(* IEC 61131-3 sources: AXOpen/src/components.dukane.welders/ctrl/src/Axo_IQ_SeriesWelder (part 4) *)

            array_buffer[169].%X0 := buf5.LimitWeld1EnergyEnable._8;
            array_buffer[169].%X1 := buf5.LimitWeld1EnergyEnable._9;
            array_buffer[169].%X2 := buf5.LimitWeld1EnergyEnable._10;
            array_buffer[169].%X3 := buf5.LimitWeld1EnergyEnable._11;
            array_buffer[169].%X4 := buf5.LimitWeld1EnergyEnable._12;
            array_buffer[169].%X5 := buf5.LimitWeld1EnergyEnable._13;
            array_buffer[169].%X6 := buf5.LimitWeld1EnergyEnable._14;
            array_buffer[169].%X7 := buf5.LimitWeld1EnergyEnable._15;

            array_buffer[170].%X0 := buf5.LimitWeld1EnergyEnable._16;
            array_buffer[170].%X1 := buf5.LimitWeld1EnergyEnable._17;
            array_buffer[170].%X2 := buf5.LimitWeld1EnergyEnable._18;
            array_buffer[170].%X3 := buf5.LimitWeld1EnergyEnable._19;
            array_buffer[170].%X4 := buf5.LimitWeld1EnergyEnable._20;
            array_buffer[170].%X5 := buf5.LimitWeld1EnergyEnable._21;
            array_buffer[170].%X6 := buf5.LimitWeld1EnergyEnable._22;
            array_buffer[170].%X7 := buf5.LimitWeld1EnergyEnable._23;

            array_buffer[171].%X0 := buf5.LimitWeld1EnergyEnable.LowerBad_1;
            array_buffer[171].%X1 := buf5.LimitWeld1EnergyEnable.LowerSuspect_1;
            array_buffer[171].%X2 := buf5.LimitWeld1EnergyEnable.UpperSuspect_1;
            array_buffer[171].%X3 := buf5.LimitWeld1EnergyEnable.UpperBad_1;
            array_buffer[171].%X4 := buf5.LimitWeld1EnergyEnable.Display_1;
            array_buffer[171].%X5 := buf5.LimitWeld1EnergyEnable._29;
            array_buffer[171].%X6 := buf5.LimitWeld1EnergyEnable._30;
            array_buffer[171].%X7 := buf5.LimitWeld1EnergyEnable._31;

            // --- LimitWeld1PowerEnable bits (bytes 172..175) ---
            array_buffer[172].%X0 := buf5.LimitWeld1PowerEnable._0;
            array_buffer[172].%X1 := buf5.LimitWeld1PowerEnable._1;
            array_buffer[172].%X2 := buf5.LimitWeld1PowerEnable._2;
            array_buffer[172].%X3 := buf5.LimitWeld1PowerEnable._3;
            array_buffer[172].%X4 := buf5.LimitWeld1PowerEnable._4;
            array_buffer[172].%X5 := buf5.LimitWeld1PowerEnable._5;
            array_buffer[172].%X6 := buf5.LimitWeld1PowerEnable._6;
            array_buffer[172].%X7 := buf5.LimitWeld1PowerEnable._7;

            array_buffer[173].%X0 := buf5.LimitWeld1PowerEnable._8;
            array_buffer[173].%X1 := buf5.LimitWeld1PowerEnable._9;
            array_buffer[173].%X2 := buf5.LimitWeld1PowerEnable._10;
            array_buffer[173].%X3 := buf5.LimitWeld1PowerEnable._11;
            array_buffer[173].%X4 := buf5.LimitWeld1PowerEnable._12;
            array_buffer[173].%X5 := buf5.LimitWeld1PowerEnable._13;
            array_buffer[173].%X6 := buf5.LimitWeld1PowerEnable._14;
            array_buffer[173].%X7 := buf5.LimitWeld1PowerEnable._15;

            array_buffer[174].%X0 := buf5.LimitWeld1PowerEnable._16;
            array_buffer[174].%X1 := buf5.LimitWeld1PowerEnable._17;
            array_buffer[174].%X2 := buf5.LimitWeld1PowerEnable._18;
            array_buffer[174].%X3 := buf5.LimitWeld1PowerEnable._19;
            array_buffer[174].%X4 := buf5.LimitWeld1PowerEnable._20;
            array_buffer[174].%X5 := buf5.LimitWeld1PowerEnable._21;
            array_buffer[174].%X6 := buf5.LimitWeld1PowerEnable._22;
            array_buffer[174].%X7 := buf5.LimitWeld1PowerEnable._23;

            array_buffer[175].%X0 := buf5.LimitWeld1PowerEnable.LowerBad_1;
            array_buffer[175].%X1 := buf5.LimitWeld1PowerEnable.LowerSuspect_1;
            array_buffer[175].%X2 := buf5.LimitWeld1PowerEnable.UpperSuspect_1;
            array_buffer[175].%X3 := buf5.LimitWeld1PowerEnable.UpperBad_1;
            array_buffer[175].%X4 := buf5.LimitWeld1PowerEnable.Display_1;
            array_buffer[175].%X5 := buf5.LimitWeld1PowerEnable._29;
            array_buffer[175].%X6 := buf5.LimitWeld1PowerEnable._30;
            array_buffer[175].%X7 := buf5.LimitWeld1PowerEnable._31;

        END_METHOD

        ///<summary>
        /// Runs tasks and logic of this component.
        /// >[!IMPORTANT] This method must or one of its overloads be called cyclically.
        ///</summary>
        METHOD PUBLIC Run
            VAR_INPUT
                parent      :   IAxoObject;
                hwID        :   UINT;
            END_VAR

            VAR_TEMP
                prev_rd_req : Bool;
                rd_any_response : Bool;
                tmp_bit : Bool;
                prev_wr_req : Bool;
                wr_any_response : Bool;
                mask : Word;
                tmp_W : Word;
                tmp_DW : DWord;
                _data_in      :   ARRAY[0..139] OF BYTE;
                _data_out     :   ARRAY[0..19] OF BYTE;
                _data_255 : ARRAY[0..254] OF BYTE;
                index : UINT;
            END_VAR

            // IQ ULTRASONIC GENERATOR CONTROL - over profinet - mode "Profinet with Distance"
            // Created by: Vaclav Fiala (fiala@gfm.cz)
            // Rewrited 1-to-1 to SCL by Tomas Kovac

            // ============================================================================
            // Adapted from original example code BY Dukane TO make the multi
            // INSTANCE use easier TO deploy AND less error prone.
            // NOTE:  use the IQ Commander software (connected over USB TO the Generator)
            // TO set the comunicatiom mode TO "Profinet with Distance" -
            // otherwise the communication will NOT work.

            // ============================================================================

            SUPER.Run(parent);

            Messenger.Serve(THIS);

            Progress := _progress;

            IF NOT _initHwCheckDone THEN
                IF parent = NULL THEN
                    Messenger.Activate(UINT#700, eAxoMessageCategory#ProgrammingError);
                    Status.Error.Id := UINT#700;
                    RETURN;
                END_IF;
                IF hwID = UINT#0 THEN
                    Messenger.Activate(UINT#701, eAxoMessageCategory#ProgrammingError);
                    Status.Error.Id := UINT#701;
                    RETURN;
                END_IF;

                Config.HWIDs.HW_Device := hwID;
                _retval := ReadSlotFromHardwareID(hardwareID := Config.HWIDs.HW_Device, geoAddr :=_geoAddr);
                IF _retval = WORD#8090 THEN
                    Messenger.Activate(UINT#702,eAxoMessageCategory#Error);
                    Status.Error.Id := UINT#702;
                    RETURN;
                END_IF;

                //******************Slot 1*****************//
                _geoAddr.Slot   :=  UINT#1;
                _geoAddr.HardwareType := UINT#4; // (4-Module)
                _retval := ReadHardwareIDFromSlot(geoAddr := _geoAddr, hardwareID => Config.HWIDs.HwID_iQ_to_PLC_Inputs);
                IF Config.HWIDs.HwID_iQ_to_PLC_Inputs = UINT#0 THEN
                    Messenger.Activate(UINT#710,eAxoMessageCategory#Error);
                    Status.Error.Id := UINT#710;
                    RETURN;
                END_IF;
                IF _retval = WORD#8091 THEN
                    Messenger.Activate(UINT#711,eAxoMessageCategory#Error);
                    Status.Error.Id := UINT#711;
                    RETURN;
                END_IF;
                IF _retval = WORD#8094 THEN
                    Messenger.Activate(UINT#712,eAxoMessageCategory#Error);
                    Status.Error.Id := UINT#712;
                    RETURN;
                END_IF;
                IF _retval = WORD#8095 THEN
                    Messenger.Activate(UINT#713,eAxoMessageCategory#Error);
                    Status.Error.Id := UINT#713;
                    RETURN;
                END_IF;
                IF _retval = WORD#8096 THEN
                    Messenger.Activate(UINT#714,eAxoMessageCategory#Error);
                    Status.Error.Id := UINT#714;
                    RETURN;
                END_IF;
                IF _retval = WORD#8097 THEN
                    Messenger.Activate(UINT#715,eAxoMessageCategory#Error);
                    Status.Error.Id := UINT#715;
                    RETURN;
                END_IF;
                ReadHardwareIOAddress(hardwareIdentifier :=  TO_WORD(Config.HWIDs.HwID_iQ_to_PLC_Inputs) , inputStartAddress => _inputsAddress , inputCount => _inputsCount , outputStartAddress => _outputsAddress , outputCount => _outputsCount);
                IF _inputsCount <> UINT#140 OR _outputsCount <> UINT#0 THEN
                    Messenger.Activate(UINT#716,eAxoMessageCategory#Error);
                    Status.Error.Id := UINT#716;
                    RETURN;
                END_IF;
                //******************Slot 2*****************//
                _geoAddr.Slot   :=  UINT#2;
                _geoAddr.HardwareType := UINT#4; // (4-Module)
                _retval := ReadHardwareIDFromSlot(geoAddr := _geoAddr, hardwareID => Config.HWIDs.HwID_PLC_to_iQ_Outputs);
                IF Config.HWIDs.HwID_PLC_to_iQ_Outputs = UINT#0 THEN
                    Messenger.Activate(UINT#910,eAxoMessageCategory#Error);
                    Status.Error.Id := UINT#910;
                    RETURN;
                END_IF;
                IF _retval = WORD#8091 THEN
                    Messenger.Activate(UINT#911,eAxoMessageCategory#Error);
                    Status.Error.Id := UINT#911;
                    RETURN;
                END_IF;
                IF _retval = WORD#8094 THEN
                    Messenger.Activate(UINT#912,eAxoMessageCategory#Error);
                    Status.Error.Id := UINT#912;
                    RETURN;
                END_IF;
                IF _retval = WORD#8095 THEN
                    Messenger.Activate(UINT#913,eAxoMessageCategory#Error);
                    Status.Error.Id := UINT#913;
                    RETURN;
                END_IF;
                IF _retval = WORD#8096 THEN
                    Messenger.Activate(UINT#914,eAxoMessageCategory#Error);
                    Status.Error.Id := UINT#914;
                    RETURN;
                END_IF;
                IF _retval = WORD#8097 THEN
                    Messenger.Activate(UINT#715,eAxoMessageCategory#Error);
                    Status.Error.Id := UINT#715;
                    RETURN;
                END_IF;
                ReadHardwareIOAddress(hardwareIdentifier :=  TO_WORD(Config.HWIDs.HwID_PLC_to_iQ_Outputs) , inputStartAddress => _inputsAddress , inputCount => _inputsCount , outputStartAddress => _outputsAddress , outputCount => _outputsCount);
                IF _outputsCount <> UINT#20 OR _inputsCount <> UINT#0 THEN
                    Messenger.Activate(UINT#916,eAxoMessageCategory#Error);
                    Status.Error.Id := UINT#916;
                    RETURN;
                END_IF;

                IF parent = NULL THEN
                    Messenger.Activate(UINT#1130,eAxoMessageCategory#Error);
                    Status.Error.Id := UINT#1130;
                    RETURN;
                END_IF;
                IF Config.HWIDs.HW_Device  = UINT#0 THEN
                    Messenger.Activate(UINT#1131,eAxoMessageCategory#Error);
                    Status.Error.Id := UINT#1131;
                    RETURN;
                END_IF;
                IF Config.HWIDs.HwID_iQ_to_PLC_Inputs  = UINT#0 THEN
                    Messenger.Activate(UINT#1132,eAxoMessageCategory#Error);
                    Status.Error.Id := UINT#1132;
                    RETURN;
                END_IF;

                IF Config.HWIDs.HwID_PLC_to_iQ_Outputs  = UINT#0 THEN
                    Messenger.Activate(UINT#1152,eAxoMessageCategory#Error);
                    Status.Error.Id := UINT#1152;
                    RETURN;
                END_IF;

                _initHwCheckDone    := TRUE;
            END_IF;

            //***********Update inputs **************

            // ============================================================================
            // Network 1: Read synchronous data from the module (inputs)
            // ============================================================================
            // This was original inputs reading =>
            // synchronous_read_retval := DPRD_DAT(LADDR := Config.HWIDs.HwID_iQ_to_PLC_Inputs,RECORD => iq_if._in);
            // <= This was original inputs reading

            // This is new inputs reading =>
            synchronous_read_retval := TO_INT(ReadData(LADDR := TO_WORD(Config.HWIDs.HwID_iQ_to_PLC_Inputs),RECORD => _data_in));
            IF synchronous_read_retval > INT#0 THEN
                Messenger.Activate(UINT#1201, eAxoMessageCategory#ProgrammingError);
                Status.Error.Id := UINT#1201;
                RETURN;
            END_IF;
            Inputs.SystemErrorStatus.Frequency_Overload_3                    := _data_in[0].%X0;
            Inputs.SystemErrorStatus._1                                      := _data_in[0].%X1;
            Inputs.SystemErrorStatus._2                                      := _data_in[0].%X2;
            Inputs.SystemErrorStatus._3                                      := _data_in[0].%X3;
            Inputs.SystemErrorStatus.Under_Voltage_1                         := _data_in[0].%X4;
            Inputs.SystemErrorStatus._5                                      := _data_in[0].%X5;
            Inputs.SystemErrorStatus._6                                      := _data_in[0].%X6;
            Inputs.SystemErrorStatus._7                                      := _data_in[0].%X7;
            Inputs.SystemErrorStatus.Over_Amplitude_Fault                    := _data_in[1].%X0;
            Inputs.SystemErrorStatus.InternalError_5                         := _data_in[1].%X1;
            Inputs.SystemErrorStatus.US_Voltage_Overload                     := _data_in[1].%X2;
            Inputs.SystemErrorStatus._11                                     := _data_in[1].%X3;
            Inputs.SystemErrorStatus._12                                     := _data_in[1].%X4;
            Inputs.SystemErrorStatus._13                                     := _data_in[1].%X5;
            Inputs.SystemErrorStatus._14                                     := _data_in[1].%X6;
            Inputs.SystemErrorStatus._15                                     := _data_in[1].%X7;
            Inputs.SystemErrorStatus.Average_Overload                        := _data_in[2].%X0;
            Inputs.SystemErrorStatus.Current_Loop                            := _data_in[2].%X1;
            Inputs.SystemErrorStatus.Power_Not_OK                            := _data_in[2].%X2;
            Inputs.SystemErrorStatus.Over_Temperature                        := _data_in[2].%X3;
            Inputs.SystemErrorStatus._20                                     := _data_in[2].%X4;
            Inputs.SystemErrorStatus._21                                     := _data_in[2].%X5;
            Inputs.SystemErrorStatus._22                                     := _data_in[2].%X6;
            Inputs.SystemErrorStatus._23                                     := _data_in[2].%X7;
            Inputs.SystemErrorStatus.InternalError_1                         := _data_in[3].%X0;
            Inputs.SystemErrorStatus.InternalError_2                         := _data_in[3].%X1;
            Inputs.SystemErrorStatus.InternalError_3                         := _data_in[3].%X2;
            Inputs.SystemErrorStatus.InternalError_4                         := _data_in[3].%X3;
            Inputs.SystemErrorStatus.FrequencyOverload_1                     := _data_in[3].%X4;
            Inputs.SystemErrorStatus.Frequency_Overload_2                    := _data_in[3].%X5;
            Inputs.SystemErrorStatus.Peak_Overload_Positive                  := _data_in[3].%X6;
            Inputs.SystemErrorStatus.Peak_Overload_Negative                  := _data_in[3].%X7;

            tmp_DW.%B3                                                          := _data_in[4];
            tmp_DW.%B2                                                          := _data_in[5];
            tmp_DW.%B1                                                          := _data_in[6];
            tmp_DW.%B0                                                          := _data_in[7];
            Inputs.SystemInitiateError := TO_DINT(tmp_DW);

            // Inputs.SystemInitiateError := TO_DINT( SHL(TO_DWORD(_data_in[4]), UINT#24) OR SHL(TO_DWORD(_data_in[5]), UINT#16) OR SHL(TO_DWORD(_data_in[6]),  UINT#8) OR TO_DWORD(_data_in[7]));

            Inputs.SystemProcessError._0                                     := _data_in[8].%X0;
            Inputs.SystemProcessError._1                                     := _data_in[8].%X1;
            Inputs.SystemProcessError._2                                     := _data_in[8].%X2;
            Inputs.SystemProcessError._3                                     := _data_in[8].%X3;
            Inputs.SystemProcessError._4                                     := _data_in[8].%X4;
            Inputs.SystemProcessError._5                                     := _data_in[8].%X5;
            Inputs.SystemProcessError._6                                     := _data_in[8].%X6;
            Inputs.SystemProcessError._7                                     := _data_in[8].%X7;
            Inputs.SystemProcessError._8                                     := _data_in[9].%X0;
            Inputs.SystemProcessError._9                                     := _data_in[9].%X1;
            Inputs.SystemProcessError._10                                    := _data_in[9].%X2;
            Inputs.SystemProcessError._11                                    := _data_in[9].%X3;
            Inputs.SystemProcessError._12                                    := _data_in[9].%X4;
            Inputs.SystemProcessError._13                                    := _data_in[9].%X5;
            Inputs.SystemProcessError._14                                    := _data_in[9].%X6;
            Inputs.SystemProcessError._15                                    := _data_in[9].%X7;
            Inputs.SystemProcessError.Trigger_Delay                          := _data_in[10].%X0;
            Inputs.SystemProcessError.Servo_DN_Limit                         := _data_in[10].%X1;
            Inputs.SystemProcessError.Servo_TOS_Position                     := _data_in[10].%X2;
            Inputs.SystemProcessError._19                                    := _data_in[10].%X3;
            Inputs.SystemProcessError._20                                    := _data_in[10].%X4;
            Inputs.SystemProcessError._21                                    := _data_in[10].%X5;
            Inputs.SystemProcessError._22                                    := _data_in[10].%X6;
            Inputs.SystemProcessError._23                                    := _data_in[10].%X7;
            Inputs.SystemProcessError.Forced_ShutDown                        := _data_in[11].%X0;
            Inputs.SystemProcessError.Trigger_Lost_Early                     := _data_in[11].%X1;
            Inputs.SystemProcessError.Trigger_Lost_Weld                      := _data_in[11].%X2;
            Inputs.SystemProcessError.Latched_Bad_Part                       := _data_in[11].%X3;
            Inputs.SystemProcessError.PreTrigger_OverTravel                  := _data_in[11].%X4;
            Inputs.SystemProcessError.Part_Detected                          := _data_in[11].%X5;
            Inputs.SystemProcessError.PreTrigger_Time                        := _data_in[11].%X6;
            Inputs.SystemProcessError.Trigger_Time                           := _data_in[11].%X7;

            tmp_DW.%B3                                                          := _data_in[12];
            tmp_DW.%B2                                                          := _data_in[13];
            tmp_DW.%B1                                                          := _data_in[14];
            tmp_DW.%B0                                                          := _data_in[15];
            Inputs.GeneratorState := TO_DINT(tmp_DW);

            tmp_DW.%B3                                                          := _data_in[16];
            tmp_DW.%B2                                                          := _data_in[17];
            tmp_DW.%B1                                                          := _data_in[18];
            tmp_DW.%B0                                                          := _data_in[19];
            Inputs.RealTimeAmplitude := TO_DINT(tmp_DW);

            tmp_DW.%B3                                                          := _data_in[20];
            tmp_DW.%B2                                                          := _data_in[21];
            tmp_DW.%B1                                                          := _data_in[22];
            tmp_DW.%B0                                                          := _data_in[23];
            Inputs.RealTimeFrequency := TO_DINT(tmp_DW);

            tmp_DW.%B3                                                          := _data_in[24];
            tmp_DW.%B2                                                          := _data_in[25];
            tmp_DW.%B1                                                          := _data_in[26];
            tmp_DW.%B0                                                          := _data_in[27];
            Inputs.RealTimePower := TO_DINT(tmp_DW);

            Inputs.SystemStatus.res_bit24                                    := _data_in[28].%X0;
            Inputs.SystemStatus.res_bit25                                    := _data_in[28].%X1;
            Inputs.SystemStatus.res_bit26                                    := _data_in[28].%X2;
            Inputs.SystemStatus.res_bit27                                    := _data_in[28].%X3;
            Inputs.SystemStatus.res_bit28                                    := _data_in[28].%X4;
            Inputs.SystemStatus.res_bit29                                    := _data_in[28].%X5;
            Inputs.SystemStatus.res_bit30                                    := _data_in[28].%X6;
            Inputs.SystemStatus.SetupChanged                                 := _data_in[28].%X7;
            Inputs.SystemStatus.InCycle                                      := _data_in[29].%X0;
            Inputs.SystemStatus.InCycle_No_AB                                := _data_in[29].%X1;
            Inputs.SystemStatus.OverTemp                                     := _data_in[29].%X2;
            Inputs.SystemStatus.In_AfterBurst                                := _data_in[29].%X3;
            Inputs.SystemStatus.In_Test                                      := _data_in[29].%X4;
            Inputs.SystemStatus.In_TestScan                                  := _data_in[29].%X5;
            Inputs.SystemStatus.MPC_Present                                  := _data_in[29].%X6;
            Inputs.SystemStatus.res_bit23                                    := _data_in[29].%X7;
            Inputs.SystemStatus.PowerOK                                      := _data_in[30].%X0;
            Inputs.SystemStatus.MPC_Ready                                    := _data_in[30].%X1;
            Inputs.SystemStatus.Ready                                        := _data_in[30].%X2;
            Inputs.SystemStatus.Any_Fault                                    := _data_in[30].%X3;
            Inputs.SystemStatus.Overload                                     := _data_in[30].%X4;
            Inputs.SystemStatus.Estop                                        := _data_in[30].%X5;
            Inputs.SystemStatus.Online                                       := _data_in[30].%X6;
            Inputs.SystemStatus.In_Hold                                      := _data_in[30].%X7;
            Inputs.SystemStatus.Good_Part                                    := _data_in[31].%X0;
            Inputs.SystemStatus.Bad_Part                                     := _data_in[31].%X1;
            Inputs.SystemStatus.Suspect_Part                                 := _data_in[31].%X2;
            Inputs.SystemStatus.CycleStartReject                             := _data_in[31].%X3;
            Inputs.SystemStatus.Amplitude_Regulation                         := _data_in[31].%X4;
            Inputs.SystemStatus.Power_Regulation                             := _data_in[31].%X5;
            Inputs.SystemStatus.Trigger_Status                               := _data_in[31].%X6;
            Inputs.SystemStatus.US_Status                                    := _data_in[31].%X7;

            tmp_DW.%B3                                                          := _data_in[32];
            tmp_DW.%B2                                                          := _data_in[33];
            tmp_DW.%B1                                                          := _data_in[34];
            tmp_DW.%B0                                                          := _data_in[35];
            Inputs.Temperature := TO_DINT(tmp_DW);

            tmp_DW.%B3                                                          := _data_in[36];
            tmp_DW.%B2                                                          := _data_in[37];
            tmp_DW.%B1                                                          := _data_in[38];
            tmp_DW.%B0                                                          := _data_in[39];
            Inputs.CycleCount := TO_DINT(tmp_DW);

            tmp_DW.%B3                                                          := _data_in[40];
            tmp_DW.%B2                                                          := _data_in[41];
            tmp_DW.%B1                                                          := _data_in[42];
            tmp_DW.%B0                                                          := _data_in[43];
            Inputs.GoodPartCount := TO_DINT(tmp_DW);

            tmp_DW.%B3                                                          := _data_in[44];
            tmp_DW.%B2                                                          := _data_in[45];
            tmp_DW.%B1                                                          := _data_in[46];
            tmp_DW.%B0                                                          := _data_in[47];
            Inputs.BadPartCount := TO_DINT(tmp_DW);

            tmp_DW.%B3                                                          := _data_in[48];
            tmp_DW.%B2                                                          := _data_in[49];
            tmp_DW.%B1                                                          := _data_in[50];
            tmp_DW.%B0                                                          := _data_in[51];
            Inputs.SuspectPartCount := TO_DINT(tmp_DW);

            tmp_DW.%B3                                                          := _data_in[52];
            tmp_DW.%B2                                                          := _data_in[53];
            tmp_DW.%B1                                                          := _data_in[54];
            tmp_DW.%B0                                                          := _data_in[55];
            Inputs.AbortedPartCount := TO_DINT(tmp_DW);

            Inputs.CyclePartStatus.LowerBadEnergyLimit                       := _data_in[56].%X0;
            Inputs.CyclePartStatus.LowerSuspectEnergyLimit                   := _data_in[56].%X1;
            Inputs.CyclePartStatus.UpperSuspectEnergyLimit                   := _data_in[56].%X2;
            Inputs.CyclePartStatus.UpperBadEnergyLimit                       := _data_in[56].%X3;
            Inputs.CyclePartStatus._4                                        := _data_in[56].%X4;
            Inputs.CyclePartStatus._5                                        := _data_in[56].%X5;
            Inputs.CyclePartStatus._6                                        := _data_in[56].%X6;
            Inputs.CyclePartStatus._7                                        := _data_in[56].%X7;
            Inputs.CyclePartStatus.LowerBadPowerLimit                        := _data_in[57].%X0;
            Inputs.CyclePartStatus.LowerSuspectPowerLimit                    := _data_in[57].%X1;
            Inputs.CyclePartStatus.UpperSuspectPowerLimit                    := _data_in[57].%X2;
            Inputs.CyclePartStatus.UpperBadPowerLimit                        := _data_in[57].%X3;
            Inputs.CyclePartStatus._12                                       := _data_in[57].%X4;
            Inputs.CyclePartStatus._13                                       := _data_in[57].%X5;
            Inputs.CyclePartStatus._14                                       := _data_in[57].%X6;
            Inputs.CyclePartStatus._15                                       := _data_in[57].%X7;
            Inputs.CyclePartStatus.LowerBadTimeLimit                         := _data_in[58].%X0;
            Inputs.CyclePartStatus.LowerSuspectTimeLimit                     := _data_in[58].%X1;
            Inputs.CyclePartStatus.UpperSuspectTimeLimit                     := _data_in[58].%X2;
            Inputs.CyclePartStatus.UpperBadTimeLimit                         := _data_in[58].%X3;
            Inputs.CyclePartStatus._20                                       := _data_in[58].%X4;
            Inputs.CyclePartStatus._21                                       := _data_in[58].%X5;
            Inputs.CyclePartStatus._22                                       := _data_in[58].%X6;
            Inputs.CyclePartStatus._23                                       := _data_in[58].%X7;
            Inputs.CyclePartStatus.GoodPart                                  := _data_in[59].%X0;
            Inputs.CyclePartStatus.BadPart                                   := _data_in[59].%X1;
            Inputs.CyclePartStatus.SuspectPart                               := _data_in[59].%X2;
            Inputs.CyclePartStatus._27                                       := _data_in[59].%X3;
            Inputs.CyclePartStatus._28                                       := _data_in[59].%X4;
            Inputs.CyclePartStatus._29                                       := _data_in[59].%X5;
            Inputs.CyclePartStatus._30                                       := _data_in[59].%X6;
            Inputs.CyclePartStatus._31                                       := _data_in[59].%X7;

            tmp_DW.%B3                                                          := _data_in[60];
            tmp_DW.%B2                                                          := _data_in[61];
            tmp_DW.%B1                                                          := _data_in[62];
            tmp_DW.%B0                                                          := _data_in[63];
            Inputs.CycleWeldTime := TO_DINT(tmp_DW);

            tmp_DW.%B3                                                          := _data_in[64];
            tmp_DW.%B2                                                          := _data_in[65];
            tmp_DW.%B1                                                          := _data_in[66];
            tmp_DW.%B0                                                          := _data_in[67];
            Inputs.CycleWeldPeakPower := TO_DINT(tmp_DW);

            tmp_DW.%B3                                                          := _data_in[68];
            tmp_DW.%B2                                                          := _data_in[69];
            tmp_DW.%B1                                                          := _data_in[70];
            tmp_DW.%B0                                                          := _data_in[71];
            Inputs.CycleWeldEnergy := TO_DINT(tmp_DW);

            tmp_DW.%B3                                                          := _data_in[72];
            tmp_DW.%B2                                                          := _data_in[73];
            tmp_DW.%B1                                                          := _data_in[74];
            tmp_DW.%B0                                                          := _data_in[75];
            Inputs.ActiveSetup := TO_DINT(tmp_DW);

            tmp_DW.%B3                                                          := _data_in[76];
            tmp_DW.%B2                                                          := _data_in[77];
            tmp_DW.%B1                                                          := _data_in[78];
            tmp_DW.%B0                                                          := _data_in[79];
            Inputs.RunningSetup := TO_DINT(tmp_DW);

            tmp_DW.%B3                                                          := _data_in[80];
            tmp_DW.%B2                                                          := _data_in[81];
            tmp_DW.%B1                                                          := _data_in[82];
            tmp_DW.%B0                                                          := _data_in[83];
            Inputs.RunningMPCProbe := TO_DINT(tmp_DW);

            tmp_DW.%B3                                                          := _data_in[84];
            tmp_DW.%B2                                                          := _data_in[85];
            tmp_DW.%B1                                                          := _data_in[86];
            tmp_DW.%B0                                                          := _data_in[87];
            Inputs.SelectedInputVoltage := TO_DINT(tmp_DW);

            tmp_DW.%B3                                                          := _data_in[88];
            tmp_DW.%B2                                                          := _data_in[89];
            tmp_DW.%B1                                                          := _data_in[90];
            tmp_DW.%B0                                                          := _data_in[91];
            Inputs.RealTimePosition := TO_DINT(tmp_DW);

            tmp_DW.%B3                                                          := _data_in[92];
            tmp_DW.%B2                                                          := _data_in[93];
            tmp_DW.%B1                                                          := _data_in[94];
            tmp_DW.%B0                                                          := _data_in[95];
            Inputs.RealTimeVelocity := TO_DINT(tmp_DW);

            Inputs.PressPartStatus_Bad_lo.Weld1Position                      := _data_in[96].%X0;
            Inputs.PressPartStatus_Bad_lo.ErrorStatus                        := _data_in[96].%X1;
            Inputs.PressPartStatus_Bad_lo._26                                := _data_in[96].%X2;
            Inputs.PressPartStatus_Bad_lo._27                                := _data_in[96].%X3;
            Inputs.PressPartStatus_Bad_lo._28                                := _data_in[96].%X4;
            Inputs.PressPartStatus_Bad_lo._29                                := _data_in[96].%X5;
            Inputs.PressPartStatus_Bad_lo._30                                := _data_in[96].%X6;
            Inputs.PressPartStatus_Bad_lo._31                                := _data_in[96].%X7;
            Inputs.PressPartStatus_Bad_lo.TotalWeldTime                      := _data_in[97].%X0;
            Inputs.PressPartStatus_Bad_lo.TotalWeldDistance                  := _data_in[97].%X1;
            Inputs.PressPartStatus_Bad_lo.TotalWeldEnergy                    := _data_in[97].%X2;
            Inputs.PressPartStatus_Bad_lo.HoldTime                           := _data_in[97].%X3;
            Inputs.PressPartStatus_Bad_lo.HoldDistance                       := _data_in[97].%X4;
            Inputs.PressPartStatus_Bad_lo.TotalCycleTime                     := _data_in[97].%X5;
            Inputs.PressPartStatus_Bad_lo.FinalHoldPosition                  := _data_in[97].%X6;
            Inputs.PressPartStatus_Bad_lo.Weld1PeakForce                     := _data_in[97].%X7;
            Inputs.PressPartStatus_Bad_lo.Weld1Distance                      := _data_in[98].%X0;
            Inputs.PressPartStatus_Bad_lo.Weld1Energy                        := _data_in[98].%X1;
            Inputs.PressPartStatus_Bad_lo.Weld1Power                         := _data_in[98].%X2;
            Inputs.PressPartStatus_Bad_lo.Weld2Time                          := _data_in[98].%X3;
            Inputs.PressPartStatus_Bad_lo.Weld2Distance                      := _data_in[98].%X4;
            Inputs.PressPartStatus_Bad_lo.Weld2Energy                        := _data_in[98].%X5;
            Inputs.PressPartStatus_Bad_lo.Weld2Power                         := _data_in[98].%X6;
            Inputs.PressPartStatus_Bad_lo.Weld2Position                      := _data_in[98].%X7;
            Inputs.PressPartStatus_Bad_lo.TriggerTime                        := _data_in[99].%X0;
            Inputs.PressPartStatus_Bad_lo.TriggerPosition                    := _data_in[99].%X1;
            Inputs.PressPartStatus_Bad_lo.AverageSensingVelocity             := _data_in[99].%X2;
            Inputs.PressPartStatus_Bad_lo.TriggerPressure                    := _data_in[99].%X3;
            Inputs.PressPartStatus_Bad_lo.TriggerForce                       := _data_in[99].%X4;
            Inputs.PressPartStatus_Bad_lo.TriggerDelayTime                   := _data_in[99].%X5;
            Inputs.PressPartStatus_Bad_lo.TriggerDelayDistance               := _data_in[99].%X6;
            Inputs.PressPartStatus_Bad_lo.Weld1Time                          := _data_in[99].%X7;

            Inputs.PressPartStatus_Sus_lo.Weld1Position                      := _data_in[100].%X0;
            Inputs.PressPartStatus_Sus_lo.ErrorStatus                        := _data_in[100].%X1;
            Inputs.PressPartStatus_Sus_lo._26                                := _data_in[100].%X2;
            Inputs.PressPartStatus_Sus_lo._27                                := _data_in[100].%X3;
            Inputs.PressPartStatus_Sus_lo._28                                := _data_in[100].%X4;
            Inputs.PressPartStatus_Sus_lo._29                                := _data_in[100].%X5;
            Inputs.PressPartStatus_Sus_lo._30                                := _data_in[100].%X6;
            Inputs.PressPartStatus_Sus_lo._31                                := _data_in[100].%X7;
            Inputs.PressPartStatus_Sus_lo.TotalWeldTime                      := _data_in[101].%X0;
            Inputs.PressPartStatus_Sus_lo.TotalWeldDistance                  := _data_in[101].%X1;
            Inputs.PressPartStatus_Sus_lo.TotalWeldEnergy                    := _data_in[101].%X2;
            Inputs.PressPartStatus_Sus_lo.HoldTime                           := _data_in[101].%X3;
            Inputs.PressPartStatus_Sus_lo.HoldDistance                       := _data_in[101].%X4;
            Inputs.PressPartStatus_Sus_lo.TotalCycleTime                     := _data_in[101].%X5;
            Inputs.PressPartStatus_Sus_lo.FinalHoldPosition                  := _data_in[101].%X6;
            Inputs.PressPartStatus_Sus_lo.Weld1PeakForce                     := _data_in[101].%X7;
            Inputs.PressPartStatus_Sus_lo.Weld1Distance                      := _data_in[102].%X0;
            Inputs.PressPartStatus_Sus_lo.Weld1Energy                        := _data_in[102].%X1;
            Inputs.PressPartStatus_Sus_lo.Weld1Power                         := _data_in[102].%X2;
            Inputs.PressPartStatus_Sus_lo.Weld2Time                          := _data_in[102].%X3;
            Inputs.PressPartStatus_Sus_lo.Weld2Distance                      := _data_in[102].%X4;
            Inputs.PressPartStatus_Sus_lo.Weld2Energy                        := _data_in[102].%X5;
            Inputs.PressPartStatus_Sus_lo.Weld2Power                         := _data_in[102].%X6;
            Inputs.PressPartStatus_Sus_lo.Weld2Position                      := _data_in[102].%X7;
            Inputs.PressPartStatus_Sus_lo.TriggerTime                        := _data_in[103].%X0;
            Inputs.PressPartStatus_Sus_lo.TriggerPosition                    := _data_in[103].%X1;
            Inputs.PressPartStatus_Sus_lo.AverageSensingVelocity             := _data_in[103].%X2;
            Inputs.PressPartStatus_Sus_lo.TriggerPressure                    := _data_in[103].%X3;
            Inputs.PressPartStatus_Sus_lo.TriggerForce                       := _data_in[103].%X4;
            Inputs.PressPartStatus_Sus_lo.TriggerDelayTime                   := _data_in[103].%X5;
            Inputs.PressPartStatus_Sus_lo.TriggerDelayDistance               := _data_in[103].%X6;
            Inputs.PressPartStatus_Sus_lo.Weld1Time                          := _data_in[103].%X7;

            Inputs.PressPartStatus_Sus_hi.Weld1Position                      := _data_in[104].%X0;
            Inputs.PressPartStatus_Sus_hi.ErrorStatus                        := _data_in[104].%X1;
            Inputs.PressPartStatus_Sus_hi._26                                := _data_in[104].%X2;
            Inputs.PressPartStatus_Sus_hi._27                                := _data_in[104].%X3;
            Inputs.PressPartStatus_Sus_hi._28                                := _data_in[104].%X4;
            Inputs.PressPartStatus_Sus_hi._29                                := _data_in[104].%X5;
            Inputs.PressPartStatus_Sus_hi._30                                := _data_in[104].%X6;
            Inputs.PressPartStatus_Sus_hi._31                                := _data_in[104].%X7;
            Inputs.PressPartStatus_Sus_hi.TotalWeldTime                      := _data_in[105].%X0;
            Inputs.PressPartStatus_Sus_hi.TotalWeldDistance                  := _data_in[105].%X1;
            Inputs.PressPartStatus_Sus_hi.TotalWeldEnergy                    := _data_in[105].%X2;
            Inputs.PressPartStatus_Sus_hi.HoldTime                           := _data_in[105].%X3;
            Inputs.PressPartStatus_Sus_hi.HoldDistance                       := _data_in[105].%X4;
            Inputs.PressPartStatus_Sus_hi.TotalCycleTime                     := _data_in[105].%X5;
            Inputs.PressPartStatus_Sus_hi.FinalHoldPosition                  := _data_in[105].%X6;
            Inputs.PressPartStatus_Sus_hi.Weld1PeakForce                     := _data_in[105].%X7;
            Inputs.PressPartStatus_Sus_hi.Weld1Distance                      := _data_in[106].%X0;
            Inputs.PressPartStatus_Sus_hi.Weld1Energy                        := _data_in[106].%X1;
            Inputs.PressPartStatus_Sus_hi.Weld1Power                         := _data_in[106].%X2;
            Inputs.PressPartStatus_Sus_hi.Weld2Time                          := _data_in[106].%X3;
            Inputs.PressPartStatus_Sus_hi.Weld2Distance                      := _data_in[106].%X4;
            Inputs.PressPartStatus_Sus_hi.Weld2Energy                        := _data_in[106].%X5;
            Inputs.PressPartStatus_Sus_hi.Weld2Power                         := _data_in[106].%X6;
            Inputs.PressPartStatus_Sus_hi.Weld2Position                      := _data_in[106].%X7;
            Inputs.PressPartStatus_Sus_hi.TriggerTime                        := _data_in[107].%X0;
            Inputs.PressPartStatus_Sus_hi.TriggerPosition                    := _data_in[107].%X1;
            Inputs.PressPartStatus_Sus_hi.AverageSensingVelocity             := _data_in[107].%X2;
            Inputs.PressPartStatus_Sus_hi.TriggerPressure                    := _data_in[107].%X3;
            Inputs.PressPartStatus_Sus_hi.TriggerForce                       := _data_in[107].%X4;
            Inputs.PressPartStatus_Sus_hi.TriggerDelayTime                   := _data_in[107].%X5;
            Inputs.PressPartStatus_Sus_hi.TriggerDelayDistance               := _data_in[107].%X6;
            Inputs.PressPartStatus_Sus_hi.Weld1Time                          := _data_in[107].%X7;

            Inputs.PressPartStatus_Bad_hi.Weld1Position                      := _data_in[108].%X0;
            Inputs.PressPartStatus_Bad_hi.ErrorStatus                        := _data_in[108].%X1;
            Inputs.PressPartStatus_Bad_hi._26                                := _data_in[108].%X2;
            Inputs.PressPartStatus_Bad_hi._27                                := _data_in[108].%X3;
            Inputs.PressPartStatus_Bad_hi._28                                := _data_in[108].%X4;
            Inputs.PressPartStatus_Bad_hi._29                                := _data_in[108].%X5;
            Inputs.PressPartStatus_Bad_hi._30                                := _data_in[108].%X6;
            Inputs.PressPartStatus_Bad_hi._31                                := _data_in[108].%X7;
            Inputs.PressPartStatus_Bad_hi.TotalWeldTime                      := _data_in[109].%X0;
            Inputs.PressPartStatus_Bad_hi.TotalWeldDistance                  := _data_in[109].%X1;
            Inputs.PressPartStatus_Bad_hi.TotalWeldEnergy                    := _data_in[109].%X2;
            Inputs.PressPartStatus_Bad_hi.HoldTime                           := _data_in[109].%X3;
            Inputs.PressPartStatus_Bad_hi.HoldDistance                       := _data_in[109].%X4;
            Inputs.PressPartStatus_Bad_hi.TotalCycleTime                     := _data_in[109].%X5;
            Inputs.PressPartStatus_Bad_hi.FinalHoldPosition                  := _data_in[109].%X6;
            Inputs.PressPartStatus_Bad_hi.Weld1PeakForce                     := _data_in[109].%X7;
            Inputs.PressPartStatus_Bad_hi.Weld1Distance                      := _data_in[110].%X0;
            Inputs.PressPartStatus_Bad_hi.Weld1Energy                        := _data_in[110].%X1;
            Inputs.PressPartStatus_Bad_hi.Weld1Power                         := _data_in[110].%X2;
            Inputs.PressPartStatus_Bad_hi.Weld2Time                          := _data_in[110].%X3;
            Inputs.PressPartStatus_Bad_hi.Weld2Distance                      := _data_in[110].%X4;
            Inputs.PressPartStatus_Bad_hi.Weld2Energy                        := _data_in[110].%X5;
            Inputs.PressPartStatus_Bad_hi.Weld2Power                         := _data_in[110].%X6;
            Inputs.PressPartStatus_Bad_hi.Weld2Position                      := _data_in[110].%X7;
            Inputs.PressPartStatus_Bad_hi.TriggerTime                        := _data_in[111].%X0;
            Inputs.PressPartStatus_Bad_hi.TriggerPosition                    := _data_in[111].%X1;
            Inputs.PressPartStatus_Bad_hi.AverageSensingVelocity             := _data_in[111].%X2;
            Inputs.PressPartStatus_Bad_hi.TriggerPressure                    := _data_in[111].%X3;
            Inputs.PressPartStatus_Bad_hi.TriggerForce                       := _data_in[111].%X4;
            Inputs.PressPartStatus_Bad_hi.TriggerDelayTime                   := _data_in[111].%X5;
            Inputs.PressPartStatus_Bad_hi.TriggerDelayDistance               := _data_in[111].%X6;
            Inputs.PressPartStatus_Bad_hi.Weld1Time                          := _data_in[111].%X7;

            tmp_DW.%B3                                                          := _data_in[112];
            tmp_DW.%B2                                                          := _data_in[113];
            tmp_DW.%B1                                                          := _data_in[114];
            tmp_DW.%B0                                                          := _data_in[115];
            Inputs.CycleTriggerTime := TO_DINT(tmp_DW);

            tmp_DW.%B3                                                          := _data_in[116];
            tmp_DW.%B2                                                          := _data_in[117];
            tmp_DW.%B1                                                          := _data_in[118];
            tmp_DW.%B0                                                          := _data_in[119];
            Inputs.CycleTriggerPosition := TO_DINT(tmp_DW);

            tmp_DW.%B3                                                          := _data_in[120];
            tmp_DW.%B2                                                          := _data_in[121];
            tmp_DW.%B1                                                          := _data_in[122];
            tmp_DW.%B0                                                          := _data_in[123];
            Inputs.CycleTriggerDelayTime := TO_DINT(tmp_DW);

            tmp_DW.%B3                                                          := _data_in[124];
            tmp_DW.%B2                                                          := _data_in[125];
            tmp_DW.%B1                                                          := _data_in[126];
            tmp_DW.%B0                                                          := _data_in[127];
            Inputs.CycleTriggerDelayDistance := TO_DINT(tmp_DW);

            tmp_DW.%B3                                                          := _data_in[128];
            tmp_DW.%B2                                                          := _data_in[129];
            tmp_DW.%B1                                                          := _data_in[130];
            tmp_DW.%B0                                                          := _data_in[131];
            Inputs.CycleWeld1Distance := TO_DINT(tmp_DW);

            tmp_DW.%B3                                                          := _data_in[132];
            tmp_DW.%B2                                                          := _data_in[133];
            tmp_DW.%B1                                                          := _data_in[134];
            tmp_DW.%B0                                                          := _data_in[135];
            Inputs.CycleWeld1Position := TO_DINT(tmp_DW);

            tmp_DW.%B3                                                          := _data_in[136];
            tmp_DW.%B2                                                          := _data_in[137];
            tmp_DW.%B1                                                          := _data_in[138];
            tmp_DW.%B0                                                          := _data_in[139];
            Inputs.CycleTotalTime := TO_DINT(tmp_DW);
            // <= This is new inputs reading

            //*****************************************
            coms_read_ok := (synchronous_read_retval = 0);

            // HMI sync OK flag
            Hmi.s.ComsSyncReadOK := coms_stable;

            // qualify stable comms (no sync errors for 1s)
            // ton_coms_stable(IN := coms_read_ok, PT := T#1s);
            // coms_stable := ton_coms_stable.Q;
            ton_coms_stable(signal := coms_read_ok, duration := T#1s);
            coms_stable := ton_coms_stable.output;

            // rising edge of comms restored
            coms_just_restored := coms_stable AND (NOT p_coms_stable);
            p_coms_stable := coms_stable;

            // ============================================================================
            // Network 2: Clear model info on lost coms
            // ============================================================================

            // IF NOT coms_read_ok THEN
            //     ModelInfo.ModelNumber := '';
            //     ModelInfo.SerialNumber := DINT#0;
            //     ModelInfo.MB_FirmwareVersion := '';
            //     ModelInfo.FP_FirmwareVersion := '';
            //     ModelInfo.MB_BootLoaderVersion := '';
            //     ModelInfo.FP_BootloaderVersion := '';
            // END_IF;

            // ============================================================================
            // Network 3: Initialize read request
            // ============================================================================

            IF coms_just_restored OR coms_stable AND AxoTaskRefresh THEN
                model_read_map := initial_model_refresh;
                par_read_map := initial_parameter_refresh;
                AxoTaskRefresh := FALSE;
            END_IF;

            // ============================================================================
            // Network 4: Process synchronous data into HMI status
            // ============================================================================

            Hmi.s.RunningAndActiveSetupNotSame := (Inputs.ActiveSetup <> Inputs.RunningSetup);

            // ============================================================================
            // Network 5: To enable any other IQ control weld time must be enabled first
            // ============================================================================

            // IF Parameters.PressWeld.Weld1Source.Power OR Parameters.PressWeld.Weld1Source.Energy OR Parameters.PressWeld.Weld1Source.Distance OR
            //     Parameters.PressWeld.Weld1Source.Position OR Parameters.PressWeld.Weld1Source.Ground_Detect OR Parameters.PressWeld.Weld1Source.Force THEN
            //     Parameters.PressWeld.Weld1Source._Time := TRUE;
            // END_IF;

            // IF Parameters.PressWeld.Weld1Source.Enable_Weld_1 AND NOT pEnableWeld THEN
            //     Parameters.PressWeld.Weld1Source._Time := TRUE;
            // END_IF;
            // Parameters.PressWeld.Weld1Source.Enable_Weld_1 := Parameters.PressWeld.Weld1Source._Time;
            // pEnableWeld := Parameters.PressWeld.Weld1Source.Enable_Weld_1;

            // ============================================================================
            // Network 6: Automated reaction to (user) parameter changes
            // (handled more fully in Network 18 below - compare & set write map)
            // ============================================================================

            // IF Parameters.PressTrigger.TriggerSource.Position AND NOT pTriggerSourcePosition THEN
            //     Parameters.PressTrigger.TriggerSource.Power := FALSE;
            // END_IF;
            // pTriggerSourcePosition := Parameters.PressTrigger.TriggerSource.Position;

            // IF Parameters.PressTrigger.TriggerSource.Power AND NOT pTriggerSourcePower THEN
            //     Parameters.PressTrigger.TriggerSource.Position := FALSE;
            // END_IF;
            // pTriggerSourcePower :=Parameters.PressTrigger.TriggerSource.Power;

            // IF Parameters.PressTrigger.TriggerSource.Position AND Parameters.PressTrigger.TriggerSource.Power THEN
            //     Parameters.PressTrigger.TriggerSource.Power := FALSE;
            // END_IF;

            // Parameters.PressTrigger.TriggerSource.Enable_Trigger := Parameters.PressTrigger.TriggerSource.Position OR Parameters.PressTrigger.TriggerSource.Power;

            // Parameters.PressPretrigger.PreTriggerSource._Time := Parameters.PressTrigger.TriggerSource.Power;
            // Parameters.PressPretrigger.PreTriggerSource.Enable_Trigger := Parameters.PressTrigger.TriggerSource.Power;
            // IF Parameters.PressTrigger.TriggerSource.Power THEN
            //     Parameters.PressPretrigger.PreTriggerTime := 0;
            // END_IF;

            // ============================================================================
            // Network 7: Afterburst enable / disable (handled via buf5 fields)
            // ============================================================================
            // tmp_DW := TO_DWORD(Parameters.AfterburstEnable) AND DWORD#1;
            // IF tmp_DW <> DWORD#0 THEN
            //     Parameters.AfterburstEnable := TO_DINT(TO_DWORD(Parameters.AfterburstEnable) OR DWORD#2);
            // ELSE
            //     Parameters.AfterburstEnable := DINT#0;
            // END_IF;

            // ============================================================================
            // Network 8: HMI processing (user controls -> request bits)
            // ============================================================================
            // IF Hmi.c.flip_freq_tracking_compat THEN
            //     Hmi.c.flip_freq_tracking_compat := FALSE;
            //     tmp_bit := (Parameters.FreqCtrlMode = 6);
            //     IF tmp_bit THEN
            //         Parameters.FreqCtrlMode := 1;
            //     ELSE
            //         Parameters.FreqCtrlMode := 0;
            //     END_IF;
            // END_IF;

            // IF Hmi.c.apply_scanned_freq THEN
            //     Hmi.c.apply_scanned_freq := FALSE;
            //     Hmi.s.DisplayApplyScannedFrequency := FALSE;
            //     IF TestScanResults.TestScanResults > 0 THEN
            //         TestScanResults.TestScanResults := TestScanResults.TestScanResults;
            //     END_IF;
            // END_IF;

            // IF Hmi.c.dont_apply_scanned_freq THEN
            //     Hmi.c.dont_apply_scanned_freq := FALSE;
            //     Hmi.s.DisplayApplyScannedFrequency := FALSE;
            //     IF Hmi.c.copy_setup THEN
            //         on_demand_write_map := on_demand_write_map OR TO_WORD(2#0000000000000001);
            //         Hmi.c.copy_setup := FALSE;
            //     END_IF;
            // END_IF;

            // ============================================================================
            // Network 9: Parameters check (safety)
            // ============================================================================
            // IF Parameters.FreqCtrlMode <> 1 AND Parameters.FreqCtrlMode <> 6 THEN
            //     Parameters.FreqCtrlMode := 1;
            // END_IF;
            // ============================================================================
            // Network 10: Trigger read on HMI req
            // ============================================================================
            IF Hmi.c.read_active_setup AND (Outputs.ActiveSetupSelection = Inputs.ActiveSetup) THEN
                par_read_map := par_read_map OR TO_WORD(2#0000000000000001);
            END_IF;

            // ============================================================================
            // Network 11: Trigger re-read on setup change indication
            // ============================================================================
            Outputs.ClearSetup := coms_read_ok AND Inputs.SystemStatus.SetupChanged;

            IF (NOT Inputs.SystemStatus.SetupChanged AND p_setup_changed) AND coms_read_ok THEN
                par_read_map := par_read_map OR initial_parameter_refresh;
            END_IF;
            p_setup_changed := Inputs.SystemStatus.SetupChanged;

            // ============================================================================
            // Network 12: Trigger test scan data read when scan finished
            // ============================================================================
            IF (NOT Inputs.SystemStatus.In_TestScan) AND p_testscan AND coms_read_ok THEN
                on_demand_read_map := on_demand_read_map OR TO_WORD(2#0000000000000001); // -> async_read_no 17
            END_IF;
            p_testscan := Inputs.SystemStatus.In_TestScan;

            // ============================================================================
            // Network 13: If Comms faulted to Generator write zeros to Generator Output.
            // ============================================================================
            //
            IF Config_reset_on_coms_fault AND NOT coms_read_ok THEN
                Outputs.RunContinuously := FALSE;
                Outputs.RunWeld := FALSE;
                Outputs.RunTest := FALSE;
                Outputs.ClearError := FALSE;
                Outputs.OTF_AmplitudeEnable := FALSE;
                Outputs.CycleStop := FALSE;
                Outputs.FrontPanelLockout_0 := FALSE;
                Outputs.FrontPanelLockout_1 := FALSE;
                Outputs.RunScan := FALSE;
                Outputs.ClearSetup := FALSE;
            END_IF;

            //*************INITIALIZATION*************
            RestoreTask.Run(THIS);
            TemplateTask_10steps_1.Run(THIS);
            TemplateTask_10steps_2.Run(THIS);
            TemplateTask_10steps_3.Run(THIS);
            TemplateTask_10steps_4.Run(THIS);
            TemplateTask_10steps_5.Run(THIS);
            TemplateTask_10steps_6.Run(THIS);
            TemplateTask_20steps_1.Run(THIS);
            TemplateTask_20steps_2.Run(THIS);
            TemplateTask_20steps_3.Run(THIS);
            TemplateTask_20steps_4.Run(THIS);
            TemplateTask_20steps_5.Run(THIS);
            TemplateTask_20steps_6.Run(THIS);

            //****************************************

            //********************Diagnostics*********
            HardwareDiagnosticsTask.Run(THIS,Config.HWIDs.HW_Device);
            //****************************************

            //*************RESTORE********************
            RestoreTask.SetIsDisabled(FALSE);
            IF RestoreTask.Execute(THIS) THEN
                THIS.Restore();
            END_IF;
            //****************************************

            //*************TemplateTask_10steps_1**************
            TemplateTask_10steps_1.SetIsDisabled(FALSE);
            IF TemplateTask_10steps_1.StartTriggered() THEN
                Status.Action.Id :=  UINT#100;
            END_IF;
            Messenger.ActivateOnCondition(ULINT#100,TemplateTask_10steps_1.IsBusy(), eAxoMessageCategory#Info);
            Messenger.ActivateOnCondition(ULINT#101,TemplateTask_10steps_1.IsDone(), eAxoMessageCategory#Info);
            IF TemplateTask_10steps_1.Execute(THIS) THEN
                IF _progress = 0 THEN
                    Status.Error.Id := UINT#0;
                    TaskMessenger.Restore();
                    THIS.CallTimers(FALSE);
                    _progress := 300;
                END_IF;

                IF _progress = 300 THEN                                                                                     // TemplateTask_10steps_1 running: , <add the detailed description of the current action 1>
                    IF _infoTimer.output THEN
                        TaskMessenger.Activate( UINT#500, eAxoMessageCategory#Warning);
                        Status.Error.Id :=      UINT#500;
                    END_IF;
                    ReadRecord2req := FALSE;
                    ReadRecord2( request := FALSE,record := str_read_buffer_254);
                    IF NOT ReadRecord2.busy AND NOT ReadRecord2.error AND NOT ReadRecord2.valid THEN
                        THIS.CallTimers(FALSE);
                        _progress := 301;
                    END_IF;
                END_IF;

                IF _progress = 301 THEN                                                                                     // TemplateTask_10steps_1 running: , <add the detailed description of the current action 2>
                    IF _infoTimer.output THEN
                        TaskMessenger.Activate( UINT#501, eAxoMessageCategory#Warning);
                        Status.Error.Id :=      UINT#501;
                    END_IF;
                    ReadRecord2maxLen := UINT#64;
                    ReadRecord2req := TRUE;
                    IF ReadRecord2.busy THEN
                        THIS.CallTimers(FALSE);
                        _progress := 302;
                    END_IF;
                END_IF;

                IF _progress = 302 THEN                                                                                     // TemplateTask_10steps_1 running: , <add the detailed description of the current action 3>
                    IF _infoTimer.output THEN
                        TaskMessenger.Activate( UINT#502, eAxoMessageCategory#Warning);
                        Status.Error.Id :=      UINT#502;
                    END_IF;

                    IF NOT ReadRecord2.busy AND ReadRecord2.valid AND NOT ReadRecord2.error THEN
                        THIS.CallTimers(FALSE);
                        _progress := 303;
                    END_IF;
                END_IF;

                IF _progress = 303 THEN                                                                                     // TemplateTask_10steps_1 running: , <add the detailed description of the current action 4>
                    IF _infoTimer.output THEN
                        TaskMessenger.Activate( UINT#503, eAxoMessageCategory#Warning);
                        Status.Error.Id :=      UINT#503;
                    END_IF;

                    IF TRUE THEN
                        THIS.CallTimers(FALSE);
                        _progress := 304;
                    END_IF;
                END_IF;

                IF _progress = 304 THEN                                                                                     // TemplateTask_10steps_1 running: , <add the detailed description of the current action 5>
                    IF _infoTimer.output THEN
                        TaskMessenger.Activate( UINT#504, eAxoMessageCategory#Warning);
                        Status.Error.Id :=      UINT#504;
                    END_IF;

                    IF TRUE THEN
                        THIS.CallTimers(FALSE);
                        _progress := 305;
                    END_IF;
                END_IF;

                IF _progress = 305 THEN                                                                                     // TemplateTask_10steps_1 running: , <add the detailed description of the current action 6>
                    IF _infoTimer.output THEN
                        TaskMessenger.Activate( UINT#505, eAxoMessageCategory#Warning);
                        Status.Error.Id :=      UINT#505;
                    END_IF;

                    IF TRUE THEN
                        THIS.CallTimers(FALSE);
                        _progress := 306;
                    END_IF;
                END_IF;

                IF _progress = 306 THEN                                                                                     // TemplateTask_10steps_1 running: , <add the detailed description of the current action 7>
                    IF _infoTimer.output THEN
                        TaskMessenger.Activate( UINT#506, eAxoMessageCategory#Warning);
                        Status.Error.Id :=      UINT#506;
                    END_IF;

                    IF TRUE THEN
                        THIS.CallTimers(FALSE);
                        _progress := 307;
                    END_IF;
                END_IF;

                IF _progress = 307 THEN                                                                                     // TemplateTask_10steps_1 running: , <add the detailed description of the current action 8>
                    IF _infoTimer.output THEN
                        TaskMessenger.Activate( UINT#507, eAxoMessageCategory#Warning);
                        Status.Error.Id :=      UINT#507;
                    END_IF;

                    IF TRUE THEN
                        THIS.CallTimers(FALSE);
                        _progress := 308;
                    END_IF;
                END_IF;

                IF _progress = 308 THEN                                                                                     // TemplateTask_10steps_1 running: , <add the detailed description of the current action 9>
                    IF _infoTimer.output THEN
                        TaskMessenger.Activate( UINT#508, eAxoMessageCategory#Warning);
                        Status.Error.Id :=      UINT#508;
                    END_IF;

                    IF TRUE THEN
                        THIS.CallTimers(FALSE);
                        _progress := 309;
                    END_IF;
                END_IF;

                IF _progress = 309 THEN
                    ReadRecord2req := FALSE;                                                                            // TemplateTask_10steps_1 running: , <add the detailed description of the current action 10>
                    TemplateTask_10steps_1.DoneWhen(TRUE);
                    _progress := 0;
                END_IF;

                ReadRecord2( request := ReadRecord2req,
                    id := TO_WORD(Config.HWIDs.HwID_iQ_to_PLC_Inputs),
                    index := index_async_model_no,
                    maxLength := ReadRecord2maxLen,
                    record := str_read_buffer_254);

                THIS.CallTimers(TRUE);

                TemplateTask_10steps_1.ThrowWhen(_errorTimer.output);
                Status.Action.Id := TO_UINT(_progress);
                TemplateTask_10steps_1.ThrowWhen(TemplateTask_10steps_1.Duration >= Config.TaskTimeout AND Config.TaskTimeout > T#0s ,'TemplateTask_10steps_1 timeout.');
            END_IF;
            IF TemplateTask_10steps_1.DoneReached() THEN
                Status.Action.Id :=  UINT#101;
                Status.Error.Id :=  UINT#0;
            ELSIF TemplateTask_10steps_1.ErrorOccured() THEN
                Status.Action.Id :=  UINT#10000;
                Status.Error.Id  :=  UINT#10000;
            ELSIF TemplateTask_10steps_1.AbortTriggered()THEN
                Status.Action.Id :=  UINT#10001;
                Status.Error.Id  :=  UINT#10001;
            END_IF;
            Messenger.ActivateOnCondition(ULINT#10000,TemplateTask_10steps_1.HasError(), eAxoMessageCategory#Error);
            Messenger.ActivateOnCondition(ULINT#10001,TemplateTask_10steps_1.IsAborted(), eAxoMessageCategory#Error);
            Messenger.ActivateOnCondition(ULINT#102,TemplateTask_10steps_1.RestoreTriggered() , eAxoMessageCategory#Error);
            IF TemplateTask_10steps_1.RestoreTriggered() AND _progress >= 300 AND _progress <= 309  THEN
                Status.Action.Id :=  UINT#102;
                _progress := 0;
            END_IF;
            //**************************************************

            //*************TemplateTask_10steps_2***************
            TemplateTask_10steps_2.SetIsDisabled(FALSE);
            IF TemplateTask_10steps_2.StartTriggered() THEN
                Status.Action.Id :=  UINT#110;
            END_IF;
            Messenger.ActivateOnCondition(ULINT#110,TemplateTask_10steps_2.IsBusy(), eAxoMessageCategory#Info);
            Messenger.ActivateOnCondition(ULINT#111,TemplateTask_10steps_2.IsDone(), eAxoMessageCategory#Info);
            IF TemplateTask_10steps_2.Execute(THIS) THEN
                IF _progress = 0 THEN
                    Status.Error.Id := UINT#0;
                    TaskMessenger.Restore();
                    THIS.CallTimers(FALSE);
                    _progress := 310;
                END_IF;

                IF _progress = 310 THEN                                                                                     // TemplateTask_10steps_2 running: , <add the detailed description of the current action 1>
                    IF _infoTimer.output THEN
                        TaskMessenger.Activate( UINT#510, eAxoMessageCategory#Warning);
                        Status.Error.Id :=      UINT#510;
                    END_IF;

                    IF TRUE THEN
                        THIS.CallTimers(FALSE);
                        _progress := 311;
                    END_IF;
                END_IF;

                IF _progress = 311 THEN                                                                                     // TemplateTask_10steps_2 running: , <add the detailed description of the current action 2>
                    IF _infoTimer.output THEN
                        TaskMessenger.Activate( UINT#511, eAxoMessageCategory#Warning);
                        Status.Error.Id :=      UINT#511;
                    END_IF;

                    IF TRUE THEN
                        THIS.CallTimers(FALSE);
                        _progress := 312;
                    END_IF;
                END_IF;

                IF _progress = 312 THEN                                                                                     // TemplateTask_10steps_2 running: , <add the detailed description of the current action 3>
                    IF _infoTimer.output THEN
                        TaskMessenger.Activate( UINT#512, eAxoMessageCategory#Warning);
                        Status.Error.Id :=      UINT#512;
                    END_IF;

                    IF TRUE THEN
                        THIS.CallTimers(FALSE);
                        _progress := 313;
                    END_IF;
                END_IF;

                IF _progress = 313 THEN                                                                                     // TemplateTask_10steps_2 running: , <add the detailed description of the current action 4>
                    IF _infoTimer.output THEN
                        TaskMessenger.Activate( UINT#513, eAxoMessageCategory#Warning);
                        Status.Error.Id :=      UINT#513;
                    END_IF;

                    IF TRUE THEN
                        THIS.CallTimers(FALSE);
                        _progress := 314;
                    END_IF;
                END_IF;

                IF _progress = 314 THEN                                                                                     // TemplateTask_10steps_2 running: , <add the detailed description of the current action 5>
                    IF _infoTimer.output THEN
                        TaskMessenger.Activate( UINT#514, eAxoMessageCategory#Warning);
                        Status.Error.Id :=      UINT#514;
                    END_IF;

                    IF TRUE THEN
                        THIS.CallTimers(FALSE);
                        _progress := 315;
                    END_IF;
                END_IF;

                IF _progress = 315 THEN                                                                                     // TemplateTask_10steps_2 running: , <add the detailed description of the current action 6>
                    IF _infoTimer.output THEN
                        TaskMessenger.Activate( UINT#515, eAxoMessageCategory#Warning);
                        Status.Error.Id :=      UINT#515;
                    END_IF;

                    IF TRUE THEN
                        THIS.CallTimers(FALSE);
                        _progress := 316;
                    END_IF;
                END_IF;

                IF _progress = 316 THEN                                                                                     // TemplateTask_10steps_2 running: , <add the detailed description of the current action 7>
                    IF _infoTimer.output THEN
                        TaskMessenger.Activate( UINT#516, eAxoMessageCategory#Warning);
                        Status.Error.Id :=      UINT#516;
                    END_IF;

                    IF TRUE THEN
                        THIS.CallTimers(FALSE);
                        _progress := 317;
                    END_IF;
                END_IF;

                IF _progress = 317 THEN                                                                                     // TemplateTask_10steps_2 running: , <add the detailed description of the current action 8>
                    IF _infoTimer.output THEN
                        TaskMessenger.Activate( UINT#517, eAxoMessageCategory#Warning);
                        Status.Error.Id :=      UINT#517;
                    END_IF;

                    IF TRUE THEN
                        THIS.CallTimers(FALSE);
                        _progress := 318;
                    END_IF;
                END_IF;

                IF _progress = 318 THEN                                                                                     // TemplateTask_10steps_2 running: , <add the detailed description of the current action 9>
                    IF _infoTimer.output THEN
                        TaskMessenger.Activate( UINT#518, eAxoMessageCategory#Warning);
                        Status.Error.Id :=      UINT#518;
                    END_IF;

                    IF TRUE THEN
                        THIS.CallTimers(FALSE);
                        _progress := 319;
                    END_IF;
                END_IF;

                IF _progress = 319 THEN                                                                                     // TemplateTask_10steps_2 running: , <add the detailed description of the current action 10>
                    TemplateTask_10steps_2.DoneWhen(TRUE);
                    _progress := 0;
                END_IF;

                THIS.CallTimers(TRUE);

                TemplateTask_10steps_2.ThrowWhen(_errorTimer.output);
                Status.Action.Id := TO_UINT(_progress);
                TemplateTask_10steps_2.ThrowWhen(TemplateTask_10steps_2.Duration >= Config.TaskTimeout AND Config.TaskTimeout > T#0s ,'TemplateTask_10steps_2 timeout.');
            END_IF;
            IF TemplateTask_10steps_2.DoneReached() THEN
                Status.Action.Id :=  UINT#111;
                Status.Error.Id :=  UINT#0;
            ELSIF TemplateTask_10steps_2.ErrorOccured() THEN
                Status.Action.Id :=  UINT#10010;
                Status.Error.Id  :=  UINT#10010;
            ELSIF TemplateTask_10steps_2.AbortTriggered()THEN
                Status.Action.Id :=  UINT#10011;
                Status.Error.Id  :=  UINT#10011;
            END_IF;
            Messenger.ActivateOnCondition(ULINT#10010,TemplateTask_10steps_2.HasError(), eAxoMessageCategory#Error);
            Messenger.ActivateOnCondition(ULINT#10011,TemplateTask_10steps_2.IsAborted(), eAxoMessageCategory#Error);
            Messenger.ActivateOnCondition(ULINT#112,TemplateTask_10steps_2.RestoreTriggered() , eAxoMessageCategory#Error);
            IF TemplateTask_10steps_2.RestoreTriggered() AND _progress >= 310 AND _progress <= 319  THEN
                Status.Action.Id :=  UINT#112;
                _progress := 0;
            END_IF;
            //**************************************************

            //*************TemplateTask_10steps_3***************
            TemplateTask_10steps_3.SetIsDisabled(FALSE);
            IF TemplateTask_10steps_3.StartTriggered() THEN
                Status.Action.Id :=  UINT#120;
            END_IF;
            Messenger.ActivateOnCondition(ULINT#120,TemplateTask_10steps_3.IsBusy(), eAxoMessageCategory#Info);
            Messenger.ActivateOnCondition(ULINT#121,TemplateTask_10steps_3.IsDone(), eAxoMessageCategory#Info);
            IF TemplateTask_10steps_3.Execute(THIS) THEN
                IF _progress = 0 THEN
                    Status.Error.Id := UINT#0;
                    TaskMessenger.Restore();
                    THIS.CallTimers(FALSE);
                    _progress := 320;
                END_IF;

                IF _progress = 320 THEN                                                                                     // TemplateTask_10steps_3 running: , <add the detailed description of the current action 1>
                    IF _infoTimer.output THEN
                        TaskMessenger.Activate( UINT#520, eAxoMessageCategory#Warning);
                        Status.Error.Id :=      UINT#520;
                    END_IF;

                    IF TRUE THEN
                        THIS.CallTimers(FALSE);
                        _progress := 321;
                    END_IF;
                END_IF;

                IF _progress = 321 THEN                                                                                     // TemplateTask_10steps_3 running: , <add the detailed description of the current action 2>
                    IF _infoTimer.output THEN
                        TaskMessenger.Activate( UINT#521, eAxoMessageCategory#Warning);
                        Status.Error.Id :=      UINT#521;
                    END_IF;

                    IF TRUE THEN
                        THIS.CallTimers(FALSE);
                        _progress := 322;
                    END_IF;
                END_IF;

                IF _progress = 322 THEN                                                                                     // TemplateTask_10steps_3 running: , <add the detailed description of the current action 3>
                    IF _infoTimer.output THEN
                        TaskMessenger.Activate( UINT#522, eAxoMessageCategory#Warning);
                        Status.Error.Id :=      UINT#522;
                    END_IF;

                    IF TRUE THEN
                        THIS.CallTimers(FALSE);
                        _progress := 323;
                    END_IF;
                END_IF;

                IF _progress = 323 THEN                                                                                     // TemplateTask_10steps_3 running: , <add the detailed description of the current action 4>
                    IF _infoTimer.output THEN
                        TaskMessenger.Activate( UINT#523, eAxoMessageCategory#Warning);
                        Status.Error.Id :=      UINT#523;
                    END_IF;

                    IF TRUE THEN
                        THIS.CallTimers(FALSE);
                        _progress := 324;
                    END_IF;
                END_IF;

                IF _progress = 324 THEN                                                                                     // TemplateTask_10steps_3 running: , <add the detailed description of the current action 5>
                    IF _infoTimer.output THEN
                        TaskMessenger.Activate( UINT#524, eAxoMessageCategory#Warning);
                        Status.Error.Id :=      UINT#524;
                    END_IF;

                    IF TRUE THEN
                        THIS.CallTimers(FALSE);
                        _progress := 325;
                    END_IF;
                END_IF;

                IF _progress = 325 THEN                                                                                     // TemplateTask_10steps_3 running: , <add the detailed description of the current action 6>
                    IF _infoTimer.output THEN
                        TaskMessenger.Activate( UINT#525, eAxoMessageCategory#Warning);
                        Status.Error.Id :=      UINT#525;
                    END_IF;

                    IF TRUE THEN
                        THIS.CallTimers(FALSE);
                        _progress := 326;
                    END_IF;
                END_IF;

                IF _progress = 326 THEN                                                                                     // TemplateTask_10steps_3 running: , <add the detailed description of the current action 7>
                    IF _infoTimer.output THEN
                        TaskMessenger.Activate( UINT#526, eAxoMessageCategory#Warning);
                        Status.Error.Id :=      UINT#526;
                    END_IF;

                    IF TRUE THEN
                        THIS.CallTimers(FALSE);
                        _progress := 327;
                    END_IF;
                END_IF;

                IF _progress = 327 THEN                                                                                     // TemplateTask_10steps_3 running: , <add the detailed description of the current action 8>
                    IF _infoTimer.output THEN
                        TaskMessenger.Activate( UINT#527, eAxoMessageCategory#Warning);
                        Status.Error.Id :=      UINT#527;
                    END_IF;

                    IF TRUE THEN
                        THIS.CallTimers(FALSE);
                        _progress := 328;
                    END_IF;
                END_IF;

                IF _progress = 328 THEN                                                                                     // TemplateTask_10steps_3 running: , <add the detailed description of the current action 9>
                    IF _infoTimer.output THEN
                        TaskMessenger.Activate( UINT#528, eAxoMessageCategory#Warning);
                        Status.Error.Id :=      UINT#528;
                    END_IF;

                    IF TRUE THEN
                        THIS.CallTimers(FALSE);
                        _progress := 329;
                    END_IF;
                END_IF;

                IF _progress = 329 THEN                                                                                     // TemplateTask_10steps_3 running: , <add the detailed description of the current action 10>
                    TemplateTask_10steps_3.DoneWhen(TRUE);
                    _progress := 0;
                END_IF;

                THIS.CallTimers(TRUE);

                TemplateTask_10steps_3.ThrowWhen(_errorTimer.output);
                Status.Action.Id := TO_UINT(_progress);
                TemplateTask_10steps_3.ThrowWhen(TemplateTask_10steps_3.Duration >= Config.TaskTimeout AND Config.TaskTimeout > T#0s ,'TemplateTask_10steps_3 timeout.');
            END_IF;
            IF TemplateTask_10steps_3.DoneReached() THEN
                Status.Action.Id :=  UINT#121;
                Status.Error.Id :=  UINT#0;
            ELSIF TemplateTask_10steps_3.ErrorOccured() THEN
                Status.Action.Id :=  UINT#10020;
                Status.Error.Id  :=  UINT#10020;
            ELSIF TemplateTask_10steps_3.AbortTriggered()THEN
                Status.Action.Id :=  UINT#10021;
                Status.Error.Id  :=  UINT#10021;
            END_IF;
            Messenger.ActivateOnCondition(ULINT#10020,TemplateTask_10steps_3.HasError(), eAxoMessageCategory#Error);
            Messenger.ActivateOnCondition(ULINT#10021,TemplateTask_10steps_3.IsAborted(), eAxoMessageCategory#Error);
            Messenger.ActivateOnCondition(ULINT#122,TemplateTask_10steps_3.RestoreTriggered() , eAxoMessageCategory#Error);
            IF TemplateTask_10steps_3.RestoreTriggered() AND _progress >= 320 AND _progress <= 329  THEN
                Status.Action.Id :=  UINT#122;
                _progress := 0;
            END_IF;
            //**************************************************

            //*************TemplateTask_10steps_4***************
            TemplateTask_10steps_4.SetIsDisabled(FALSE);
            IF TemplateTask_10steps_4.StartTriggered() THEN
                Status.Action.Id :=  UINT#130;
            END_IF;
            Messenger.ActivateOnCondition(ULINT#130,TemplateTask_10steps_4.IsBusy(), eAxoMessageCategory#Info);
            Messenger.ActivateOnCondition(ULINT#131,TemplateTask_10steps_4.IsDone(), eAxoMessageCategory#Info);
            IF TemplateTask_10steps_4.Execute(THIS) THEN
                IF _progress = 0 THEN
                    Status.Error.Id := UINT#0;
                    TaskMessenger.Restore();
                    THIS.CallTimers(FALSE);
                    _progress := 330;
                END_IF;

                IF _progress = 330 THEN                                                                                     // TemplateTask_10steps_4 running: , <add the detailed description of the current action 1>
                    IF _infoTimer.output THEN
                        TaskMessenger.Activate( UINT#530, eAxoMessageCategory#Warning);
                        Status.Error.Id :=      UINT#530;
                    END_IF;

                    IF TRUE THEN
                        THIS.CallTimers(FALSE);
                        _progress := 331;
                    END_IF;
                END_IF;

                IF _progress = 331 THEN                                                                                     // TemplateTask_10steps_4 running: , <add the detailed description of the current action 2>
                    IF _infoTimer.output THEN
                        TaskMessenger.Activate( UINT#531, eAxoMessageCategory#Warning);
                        Status.Error.Id :=      UINT#531;
                    END_IF;

                    IF TRUE THEN
                        THIS.CallTimers(FALSE);
                        _progress := 332;
                    END_IF;
                END_IF;

                IF _progress = 332 THEN                                                                                     // TemplateTask_10steps_4 running: , <add the detailed description of the current action 3>
                    IF _infoTimer.output THEN
                        TaskMessenger.Activate( UINT#532, eAxoMessageCategory#Warning);
                        Status.Error.Id :=      UINT#532;
                    END_IF;

                    IF TRUE THEN
                        THIS.CallTimers(FALSE);
                        _progress := 333;
                    END_IF;
                END_IF;

                IF _progress = 333 THEN                                                                                     // TemplateTask_10steps_4 running: , <add the detailed description of the current action 4>
                    IF _infoTimer.output THEN
                        TaskMessenger.Activate( UINT#533, eAxoMessageCategory#Warning);
                        Status.Error.Id :=      UINT#533;
                    END_IF;

                    IF TRUE THEN
                        THIS.CallTimers(FALSE);
                        _progress := 334;
                    END_IF;
                END_IF;

                IF _progress = 334 THEN                                                                                     // TemplateTask_10steps_4 running: , <add the detailed description of the current action 5>
                    IF _infoTimer.output THEN
                        TaskMessenger.Activate( UINT#534, eAxoMessageCategory#Warning);
                        Status.Error.Id :=      UINT#534;
                    END_IF;

                    IF TRUE THEN
                        THIS.CallTimers(FALSE);
                        _progress := 335;
                    END_IF;
                END_IF;

                IF _progress = 335 THEN                                                                                     // TemplateTask_10steps_4 running: , <add the detailed description of the current action 6>
                    IF _infoTimer.output THEN
                        TaskMessenger.Activate( UINT#535, eAxoMessageCategory#Warning);
                        Status.Error.Id :=      UINT#535;
                    END_IF;

                    IF TRUE THEN
                        THIS.CallTimers(FALSE);
                        _progress := 336;
                    END_IF;
                END_IF;

                IF _progress = 336 THEN                                                                                     // TemplateTask_10steps_4 running: , <add the detailed description of the current action 7>
                    IF _infoTimer.output THEN
                        TaskMessenger.Activate( UINT#536, eAxoMessageCategory#Warning);
                        Status.Error.Id :=      UINT#536;
                    END_IF;

                    IF TRUE THEN
                        THIS.CallTimers(FALSE);
                        _progress := 337;
                    END_IF;
                END_IF;

                IF _progress = 337 THEN                                                                                     // TemplateTask_10steps_4 running: , <add the detailed description of the current action 8>
                    IF _infoTimer.output THEN
                        TaskMessenger.Activate( UINT#537, eAxoMessageCategory#Warning);
                        Status.Error.Id :=      UINT#537;
                    END_IF;

                    IF TRUE THEN
                        THIS.CallTimers(FALSE);
                        _progress := 338;
                    END_IF;
                END_IF;

                IF _progress = 338 THEN                                                                                     // TemplateTask_10steps_4 running: , <add the detailed description of the current action 9>
                    IF _infoTimer.output THEN
                        TaskMessenger.Activate( UINT#538, eAxoMessageCategory#Warning);
                        Status.Error.Id :=      UINT#538;
                    END_IF;

                    IF TRUE THEN
                        THIS.CallTimers(FALSE);
                        _progress := 339;
                    END_IF;
                END_IF;

                IF _progress = 339 THEN                                                                                     // TemplateTask_10steps_4 running: , <add the detailed description of the current action 10>
                    TemplateTask_10steps_4.DoneWhen(TRUE);
                    _progress := 0;
                END_IF;

                THIS.CallTimers(TRUE);

                TemplateTask_10steps_4.ThrowWhen(_errorTimer.output);
                Status.Action.Id := TO_UINT(_progress);
                TemplateTask_10steps_4.ThrowWhen(TemplateTask_10steps_4.Duration >= Config.TaskTimeout AND Config.TaskTimeout > T#0s ,'TemplateTask_10steps_4 timeout.');
            END_IF;
            IF TemplateTask_10steps_4.DoneReached() THEN
                Status.Action.Id :=  UINT#131;
                Status.Error.Id :=  UINT#0;
            ELSIF TemplateTask_10steps_4.ErrorOccured() THEN
                Status.Action.Id :=  UINT#10030;
                Status.Error.Id  :=  UINT#10030;
            ELSIF TemplateTask_10steps_4.AbortTriggered()THEN
                Status.Action.Id :=  UINT#10031;
                Status.Error.Id  :=  UINT#10031;
            END_IF;
            Messenger.ActivateOnCondition(ULINT#10030,TemplateTask_10steps_4.HasError(), eAxoMessageCategory#Error);
            Messenger.ActivateOnCondition(ULINT#10031,TemplateTask_10steps_4.IsAborted(), eAxoMessageCategory#Error);
            Messenger.ActivateOnCondition(ULINT#132,TemplateTask_10steps_4.RestoreTriggered() , eAxoMessageCategory#Error);
            IF TemplateTask_10steps_4.RestoreTriggered() AND _progress >= 330 AND _progress <= 339  THEN
                Status.Action.Id :=  UINT#132;
                _progress := 0;
            END_IF;
            //**************************************************

            //*************TemplateTask_10steps_5***************
            TemplateTask_10steps_5.SetIsDisabled(FALSE);
            IF TemplateTask_10steps_5.StartTriggered() THEN
                Status.Action.Id :=  UINT#140;
            END_IF;
            Messenger.ActivateOnCondition(ULINT#140,TemplateTask_10steps_5.IsBusy(), eAxoMessageCategory#Info);
            Messenger.ActivateOnCondition(ULINT#141,TemplateTask_10steps_5.IsDone(), eAxoMessageCategory#Info);
            IF TemplateTask_10steps_5.Execute(THIS) THEN
                IF _progress = 0 THEN
                    Status.Error.Id := UINT#0;
                    TaskMessenger.Restore();
                    THIS.CallTimers(FALSE);
                    _progress := 340;
                END_IF;

                IF _progress = 340 THEN                                                                                     // TemplateTask_10steps_5 running: , <add the detailed description of the current action 1>
                    IF _infoTimer.output THEN
                        TaskMessenger.Activate( UINT#540, eAxoMessageCategory#Warning);
                        Status.Error.Id :=      UINT#540;
                    END_IF;
